(* Logix 5000 project; controller PRU vendor 1 type 14 code 107 rev 20.13; software revision 20.01; part 12 of 17 *)
(* tags used below, declared in another part *)
   AFI : BOOL;
   CR0_CON1_HTR1_GON : BOOL;   // ZONE 1 (L1,L2,L3)
   CR0_CON1_HTR1_LON : BOOL;   // AUTO LOGIC - ZONE 1 HEATER CONTACTOR
   CR1_CON2_HTR2_GON : BOOL;   // ZONE 2 (L1,L2,L3)
   CR1_CON2_HTR2_LON : BOOL;   // AUTO LOGIC - ZONE 2 HEATER CONTACTOR
   CR2_CON3_HTR3_GON : BOOL;   // ZONE 3 (L1,L2,L3)
   CR2_CON3_HTR3_LON : BOOL;   // AUTO LOGIC - ZONE 3 HEATER CONTACTOR
   CR3_CON4_HTR4_GON : BOOL;   // ZONE 4 (L1) ZONE 5 (L2) ZONE 6 (L3)
   CR3_CON4_HTR4_LON : BOOL;   // AUTO LOGIC - ZONES 4-6 HEATER CONTACTOR
   CR4_CON5_HTR5_GON : BOOL;   // ZONE 7 (L1) ZONE 8 (L2) ZONE 9 (L3)
   CR4_CON5_HTR5_LON : BOOL;   // AUTO LOGIC - ZONES 7-9 HEATER CONTACTOR
   CR5_CON1_SAFETY_GON : BOOL;
   CR5_CON1_SAFETY_LON : BOOL;
   CR6_CON2_SAFETY_GON : BOOL;
   CR6_CON2_SAFETY_LON : BOOL;
   CR8_VFD_DRYERR_GON : BOOL;
   CR8_VFD_DRYERR_LON : BOOL;
   ESR_CONTACT_1_ION : BOOL;
   ESR_CONTACT_2_ION : BOOL;
   ESR_RESET_PB_ION : BOOL;
   HMI_CR0_FORCE_OFF : BOOL;
   HMI_CR0_FORCE_ON : BOOL;
   HMI_CR10_FORCE_OFF : BOOL;
   HMI_CR10_FORCE_ON : BOOL;
   HMI_CR11_FORCE_OFF : BOOL;
   HMI_CR11_FORCE_ON : BOOL;
   HMI_CR12_FORCE_OFF : BOOL;
   HMI_CR12_FORCE_ON : BOOL;
   HMI_CR13_FORCE_OFF : BOOL;
   HMI_CR13_FORCE_ON : BOOL;
   HMI_CR14_FORCE_OFF : BOOL;   // Knife Gate 0621 force closed.
   HMI_CR14_FORCE_ON : BOOL;   // Knife Gate 0621 force open.
   HMI_CR15_FORCE_OFF : BOOL;   // Knife Gate 0621 force closed.
   HMI_CR15_FORCE_ON : BOOL;   // Knife Gate 0621 force open.
   HMI_CR16_FORCE_OFF : BOOL;
   HMI_CR16_FORCE_ON : BOOL;
   HMI_CR17_FORCE_OFF : BOOL;
   HMI_CR17_FORCE_ON : BOOL;
   HMI_CR19_FORCE_OFF : BOOL;
   HMI_CR19_FORCE_ON : BOOL;
   HMI_CR1_FORCE_OFF : BOOL;
   HMI_CR1_FORCE_ON : BOOL;
   HMI_CR2_FORCE_OFF : BOOL;
   HMI_CR2_FORCE_ON : BOOL;
   HMI_CR3_FORCE_OFF : BOOL;
   HMI_CR3_FORCE_ON : BOOL;
   HMI_CR4_FORCE_OFF : BOOL;
   HMI_CR4_FORCE_ON : BOOL;
   HMI_CR5_FORCE_OFF : BOOL;
   HMI_CR5_FORCE_ON : BOOL;
   HMI_CR6_FORCE_OFF : BOOL;
   HMI_CR6_FORCE_ON : BOOL;
   HMI_CR8_FORCE_OFF : BOOL;
   HMI_CR8_FORCE_ON : BOOL;
   HMI_CR9_FORCE_OFF : BOOL;
   HMI_CR9_FORCE_ON : BOOL;
   HMI_TE0101_FORCE_VALUE : INT;
   HMI_TE0101_FORCED : BOOL;
   HMI_TE0102_FORCE_VALUE : INT;
   HMI_TE0102_FORCED : BOOL;
   HMI_TE0103_FORCE_VALUE : INT;
   HMI_TE0103_FORCED : BOOL;
   HMI_TE0104_FORCE_VALUE : INT;
   HMI_TE0104_FORCED : BOOL;
   HMI_TE0105_FORCE_VALUE : INT;
   HMI_TE0105_FORCED : BOOL;
   HMI_TE0106_FORCE_VALUE : INT;
   HMI_TE0106_FORCED : BOOL;
   HMI_TE0107_FORCE_VALUE : INT;
   HMI_TE0107_FORCED : BOOL;
   HMI_TE0108_FORCE_VALUE : INT;
   HMI_TE0108_FORCED : BOOL;
   HMI_TE0109_FORCE_VALUE : DINT;
   HMI_TE0109_FORCED : BOOL;
   HMI_TE0110_FORCE_VALUE : DINT;
   HMI_TE0110_FORCED : BOOL;
   HMI_TE0111_FORCE_VALUE : DINT;
   HMI_TE0111_FORCED : BOOL;
   HMI_TE0112_FORCE_VALUE : DINT;
   HMI_TE0112_FORCED : BOOL;
   HMI_TE0113_FORCE_VALUE : DINT;
   HMI_TE0113_FORCED : BOOL;
   HMI_TE0114_FORCE_VALUE : DINT;
   HMI_TE0114_FORCED : BOOL;
   HMI_TE0115_FORCE_VALUE : DINT;
   HMI_TE0115_FORCED : BOOL;
   HMI_TE0116_FORCE_VALUE : DINT;
   HMI_TE0116_FORCED : BOOL;
   HMI_TE0117_FORCE_VALUE : DINT;
   HMI_TE0117_FORCED : BOOL;
   HMI_TE0118_FORCE_VALUE : DINT;
   HMI_TE0118_FORCED : BOOL;
   HMI_TE0119_FORCE_VALUE : DINT;
   HMI_TE0119_FORCED : BOOL;
   HMI_TE0120_FORCE_VALUE : DINT;
   HMI_TE0120_FORCED : BOOL;
   HMI_TE0121_FORCE_VALUE : DINT;
   HMI_TE0121_FORCED : BOOL;
   HMI_TE0122_FORCE_VALUE : DINT;
   HMI_TE0122_FORCED : BOOL;
   HMI_TE0123_FORCE_VALUE : DINT;
   HMI_TE0123_FORCED : BOOL;
   HMI_TE0124_FORCE_VALUE : DINT;
   HMI_TE0124_FORCED : BOOL;
   HMI_TE0125_FORCE_VALUE : DINT;
   HMI_TE0125_FORCED : BOOL;
   HMI_TE0126_FORCE_VALUE : DINT;
   HMI_TE0126_FORCED : BOOL;
   HMI_TE0127_FORCE_VALUE : DINT;
   HMI_TE0127_FORCED : BOOL;
   HMI_TE0128_FORCE_VALUE : DINT;
   HMI_TE0128_FORCED : BOOL;
   HMI_TE0129_FORCE_VALUE : DINT;
   HMI_TE0129_FORCED : BOOL;
   HMI_TE0130_FORCE_VALUE : DINT;
   HMI_TE0130_FORCED : BOOL;
   HMI_TE0201_FORCE_VALUE : DINT;
   HMI_TE0201_FORCED : BOOL;
   HMI_TE0202_FORCE_VALUE : DINT;
   HMI_TE0202_FORCED : BOOL;
   K6021_GO_CLOSE_GON : BOOL;
   K6021_GO_CLOSE_LON : BOOL;   // Knife Gate 6021 - Close Auto Logic
   K6021_GO_OPEN_GON : BOOL;
   K6021_GO_OPEN_LON : BOOL;   // Knife Gate 6021 - Open Auto Logic
   K6021_GO_STOP_GON : BOOL;
   K6022_GO_CLOSE_GON : BOOL;
   K6022_GO_CLOSE_LON : BOOL;
   K6022_GO_OPEN_GON : BOOL;
   K6022_GO_OPEN_LON : BOOL;
   K6022_GO_STOP_GON : BOOL;
   K6022_GO_STOP_LON : BOOL;
   KG021_SEQUENCER : INT;   // 1 = OPEN SV0201 2 = CLOSE SV0201 3 = OPEN KG021 4 = CLOSE KG021
   KG022_SEQUENCER : INT;   // 1 = OPEN SV0202 2 = CLOSE SV0202 3 = OPEN KG022 4 = CLOSE KG022
   PROCESS_SEQUENCER : INT;
   SHUTDOWN_PURGE_TIMER : TIMER;
   STARTUP_PURGE_TIMER : TIMER;
   SV0101 : BOOL;
   SV0101_LON : BOOL;
   SV0102 : BOOL;
   SV0102_LON : BOOL;
   SV0201 : BOOL;
   SV0201_LON : BOOL;
   SV0202 : BOOL;
   SV0202_LON : BOOL;
   SV0203 : BOOL;
   SV0203_LON : BOOL;
   TE0101 : REAL;
   TE0101_RAW : DINT;
   TE0102 : REAL;
   TE0102_RAW : DINT;
   TE0103 : REAL;
   TE0103_RAW : DINT;
   TE0104 : REAL;
   TE0104_RAW : DINT;
   TE0105 : REAL;
   TE0105_RAW : DINT;
   TE0106 : REAL;
   TE0106_RAW : DINT;
   TE0107 : REAL;
   TE0107_RAW : DINT;
   TE0108 : REAL;
   TE0108_RAW : DINT;
   TE0109 : REAL;
   TE0109_RAW : DINT;
   TE0110 : REAL;
   TE0110_RAW : DINT;
   TE0111 : REAL;
   TE0111_RAW : DINT;
   TE0112 : REAL;
   TE0112_RAW : DINT;
   TE0113 : REAL;
   TE0113_RAW : DINT;
   TE0114 : REAL;
   TE0114_RAW : DINT;
   TE0115 : REAL;
   TE0115_RAW : DINT;
   TE0116 : REAL;
   TE0116_RAW : DINT;
   TE0117 : REAL;
   TE0117_RAW : DINT;
   TE0118 : REAL;
   TE0118_RAW : DINT;
   TE0119 : REAL;
   TE0119_RAW : DINT;
   TE0120 : REAL;
   TE0120_RAW : DINT;
   TE0121 : REAL;
   TE0121_RAW : DINT;
   TE0122 : REAL;
   TE0122_RAW : DINT;
   TE0123 : REAL;
   TE0123_RAW : DINT;
   TE0124 : REAL;
   TE0124_RAW : DINT;
   TE0125 : REAL;
   TE0125_RAW : DINT;
   TE0126 : REAL;
   TE0126_RAW : DINT;
   TE0127 : REAL;
   TE0127_RAW : DINT;
   TE0128 : REAL;
   TE0128_RAW : DINT;
   TE0129 : REAL;
   TE0129_RAW : DINT;
   TE0130 : REAL;
   TE0130_RAW : DINT;
   TE0201 : REAL;
   TE0201_RAW : DINT;
   TE0202 : REAL;
   TE0202_RAW : DINT;
(* MainProgram, continued *)

ROUTINE G02_MAP_DIG_OUTPUTS   (* ladder *)
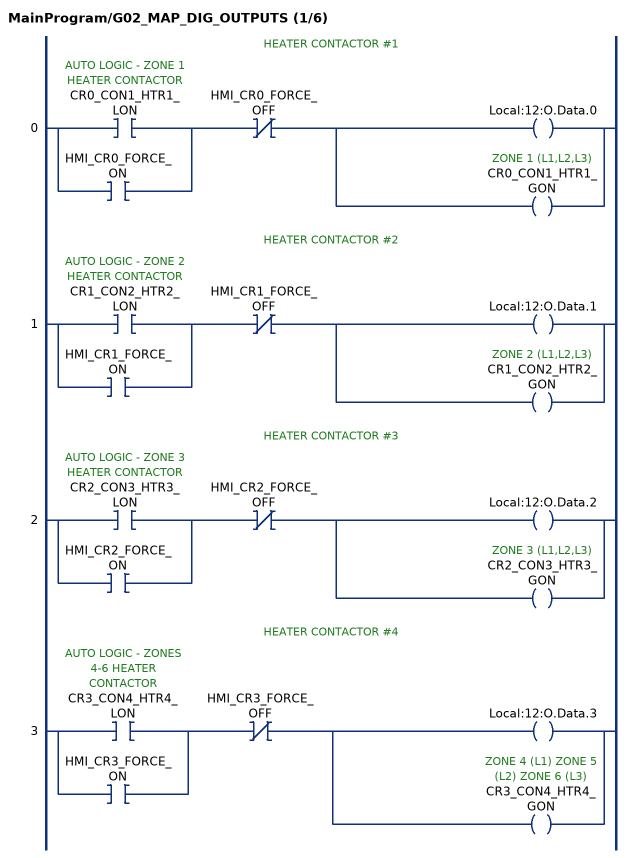
   // HEATER CONTACTOR #1
   0: [XIC(CR0_CON1_HTR1_LON) ,XIC(HMI_CR0_FORCE_ON) ]XIO(HMI_CR0_FORCE_OFF)[OTE(Local:12:O.Data.0) ,OTE(CR0_CON1_HTR1_GON) ];
   // HEATER CONTACTOR #2
   1: [XIC(CR1_CON2_HTR2_LON) ,XIC(HMI_CR1_FORCE_ON) ]XIO(HMI_CR1_FORCE_OFF)[OTE(Local:12:O.Data.1) ,OTE(CR1_CON2_HTR2_GON) ];
   // HEATER CONTACTOR #3
   2: [XIC(CR2_CON3_HTR3_LON) ,XIC(HMI_CR2_FORCE_ON) ]XIO(HMI_CR2_FORCE_OFF)[OTE(Local:12:O.Data.2) ,OTE(CR2_CON3_HTR3_GON) ];
   // HEATER CONTACTOR #4
   3: [XIC(CR3_CON4_HTR4_LON) ,XIC(HMI_CR3_FORCE_ON) ]XIO(HMI_CR3_FORCE_OFF)[OTE(Local:12:O.Data.3) ,OTE(CR3_CON4_HTR4_GON) ];
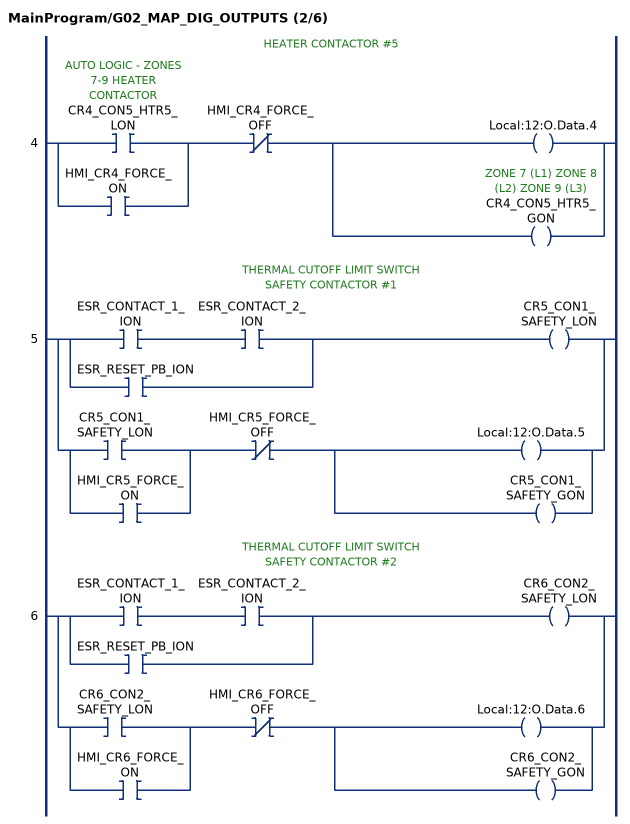
   // HEATER CONTACTOR #5
   4: [XIC(CR4_CON5_HTR5_LON) ,XIC(HMI_CR4_FORCE_ON) ]XIO(HMI_CR4_FORCE_OFF)[OTE(Local:12:O.Data.4) ,OTE(CR4_CON5_HTR5_GON) ];
   // THERMAL CUTOFF LIMIT SWITCH
   // SAFETY CONTACTOR #1
   5: [[XIC(ESR_CONTACT_1_ION) XIC(ESR_CONTACT_2_ION) ,XIC(ESR_RESET_PB_ION) ] OTE(CR5_CON1_SAFETY_LON) ,[XIC(CR5_CON1_SAFETY_LON) ,XIC(HMI_CR5_FORCE_ON) ] XIO(HMI_CR5_FORCE_OFF) [OTE(Local:12:O.Data.5) ,OTE(CR5_CON1_SAFETY_GON) ] ];
   // THERMAL CUTOFF LIMIT SWITCH
   // SAFETY CONTACTOR #2
   6: [[XIC(ESR_CONTACT_1_ION) XIC(ESR_CONTACT_2_ION) ,XIC(ESR_RESET_PB_ION) ] OTE(CR6_CON2_SAFETY_LON) ,[XIC(CR6_CON2_SAFETY_LON) ,XIC(HMI_CR6_FORCE_ON) ] XIO(HMI_CR6_FORCE_OFF) [OTE(Local:12:O.Data.6) ,OTE(CR6_CON2_SAFETY_GON) ] ];
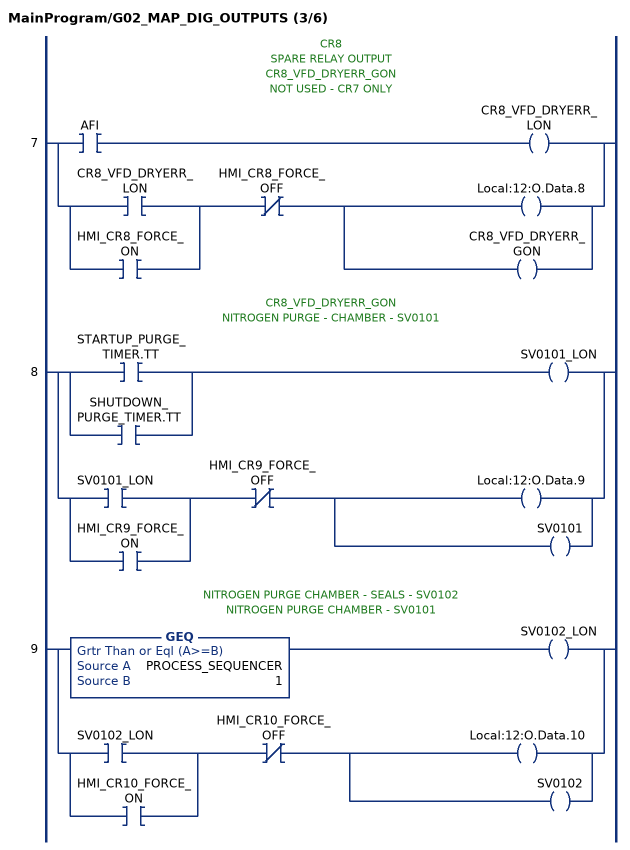
   // CR8
   // SPARE RELAY OUTPUT
   // CR8_VFD_DRYERR_GON
   // NOT USED - CR7 ONLY
   7: [XIC(AFI) OTE(CR8_VFD_DRYERR_LON) ,[XIC(CR8_VFD_DRYERR_LON) ,XIC(HMI_CR8_FORCE_ON) ] XIO(HMI_CR8_FORCE_OFF) [OTE(Local:12:O.Data.8) ,OTE(CR8_VFD_DRYERR_GON) ] ];
   // CR8_VFD_DRYERR_GON
   // NITROGEN PURGE - CHAMBER - SV0101
   8: [[XIC(STARTUP_PURGE_TIMER.TT) ,XIC(SHUTDOWN_PURGE_TIMER.TT) ] OTE(SV0101_LON) ,[XIC(SV0101_LON) ,XIC(HMI_CR9_FORCE_ON) ] XIO(HMI_CR9_FORCE_OFF) [OTE(Local:12:O.Data.9) ,OTE(SV0101) ] ];
   // NITROGEN PURGE CHAMBER - SEALS - SV0102
   // NITROGEN PURGE CHAMBER - SV0101
   9: [GEQ(PROCESS_SEQUENCER,1) OTE(SV0102_LON) ,[XIC(SV0102_LON) ,XIC(HMI_CR10_FORCE_ON) ] XIO(HMI_CR10_FORCE_OFF) [OTE(Local:12:O.Data.10) ,OTE(SV0102) ] ];
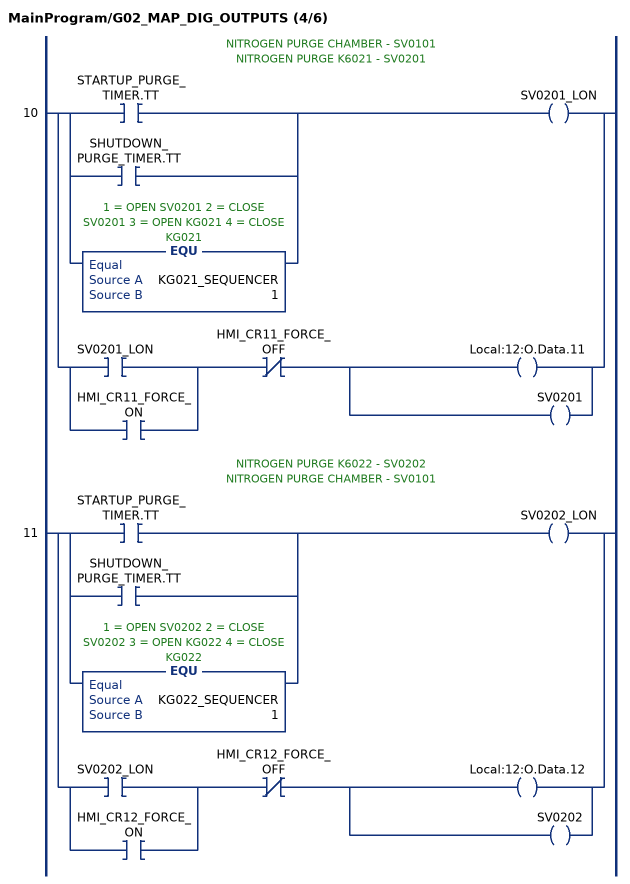
   // NITROGEN PURGE CHAMBER - SV0101
   // NITROGEN PURGE K6021 - SV0201
   10: [[XIC(STARTUP_PURGE_TIMER.TT) ,XIC(SHUTDOWN_PURGE_TIMER.TT) ,EQU(KG021_SEQUENCER,1) ] OTE(SV0201_LON) ,[XIC(SV0201_LON) ,XIC(HMI_CR11_FORCE_ON) ] XIO(HMI_CR11_FORCE_OFF) [OTE(Local:12:O.Data.11) ,OTE(SV0201) ] ];
   // NITROGEN PURGE K6022 - SV0202
   // NITROGEN PURGE CHAMBER - SV0101
   11: [[XIC(STARTUP_PURGE_TIMER.TT) ,XIC(SHUTDOWN_PURGE_TIMER.TT) ,EQU(KG022_SEQUENCER,1) ] OTE(SV0202_LON) ,[XIC(SV0202_LON) ,XIC(HMI_CR12_FORCE_ON) ] XIO(HMI_CR12_FORCE_OFF) [OTE(Local:12:O.Data.12) ,OTE(SV0202) ] ];
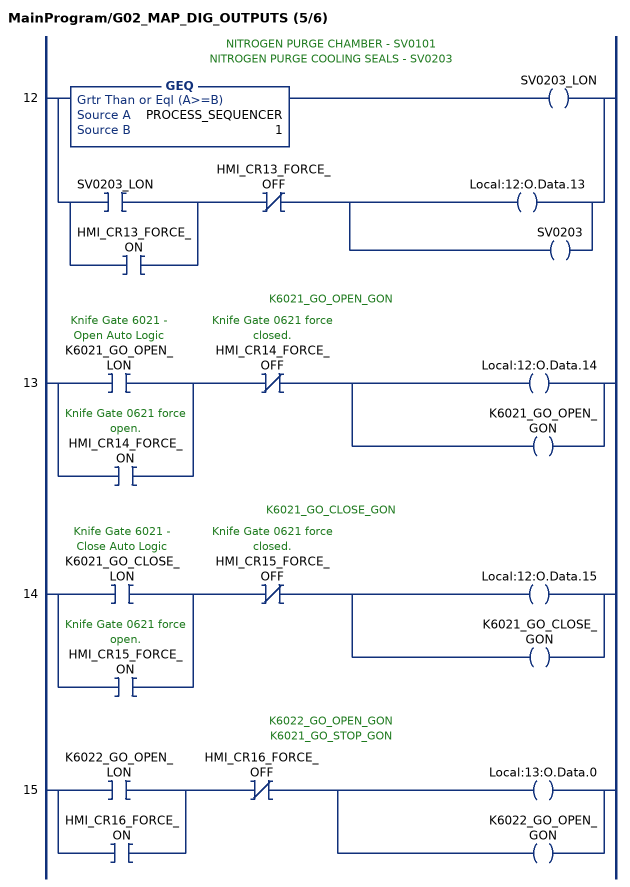
   // NITROGEN PURGE CHAMBER - SV0101
   // NITROGEN PURGE COOLING SEALS - SV0203
   12: [GEQ(PROCESS_SEQUENCER,1) OTE(SV0203_LON) ,[XIC(SV0203_LON) ,XIC(HMI_CR13_FORCE_ON) ] XIO(HMI_CR13_FORCE_OFF) [OTE(Local:12:O.Data.13) ,OTE(SV0203) ] ];
   // K6021_GO_OPEN_GON
   13: [XIC(K6021_GO_OPEN_LON) ,XIC(HMI_CR14_FORCE_ON) ]XIO(HMI_CR14_FORCE_OFF)[OTE(Local:12:O.Data.14) ,OTE(K6021_GO_OPEN_GON) ];
   // K6021_GO_CLOSE_GON
   14: [XIC(K6021_GO_CLOSE_LON) ,XIC(HMI_CR15_FORCE_ON) ]XIO(HMI_CR15_FORCE_OFF)[OTE(Local:12:O.Data.15) ,OTE(K6021_GO_CLOSE_GON) ];
   // K6022_GO_OPEN_GON
   // K6021_GO_STOP_GON
   15: [XIC(K6022_GO_OPEN_LON) ,XIC(HMI_CR16_FORCE_ON) ]XIO(HMI_CR16_FORCE_OFF)[OTE(Local:13:O.Data.0) ,OTE(K6022_GO_OPEN_GON) ];
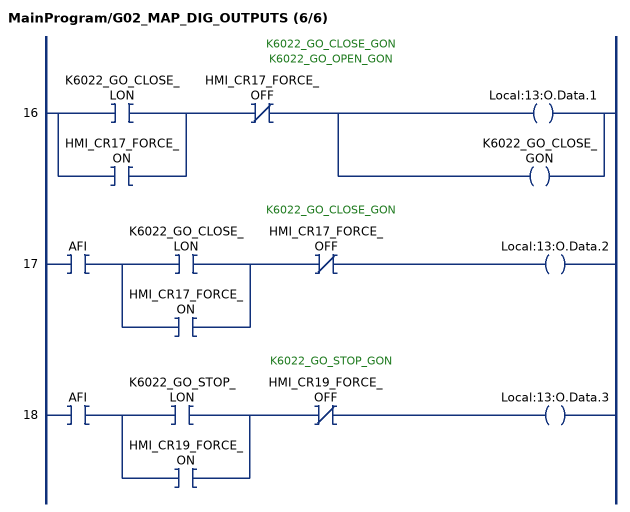
   // K6022_GO_CLOSE_GON
   // K6022_GO_OPEN_GON
   16: [XIC(K6022_GO_CLOSE_LON) ,XIC(HMI_CR17_FORCE_ON) ]XIO(HMI_CR17_FORCE_OFF)[OTE(Local:13:O.Data.1) ,OTE(K6022_GO_CLOSE_GON) ];
   // K6022_GO_CLOSE_GON
   17: XIC(AFI)[XIC(K6022_GO_CLOSE_LON) ,XIC(HMI_CR17_FORCE_ON) ]XIO(HMI_CR17_FORCE_OFF)OTE(Local:13:O.Data.2);
   // K6022_GO_STOP_GON
   18: XIC(AFI)[XIC(K6022_GO_STOP_LON) ,XIC(HMI_CR19_FORCE_ON) ]XIO(HMI_CR19_FORCE_OFF)OTE(Local:13:O.Data.3);
END_ROUTINE

ROUTINE G03_MAP_THERMOCOUPLES   (* ladder *)
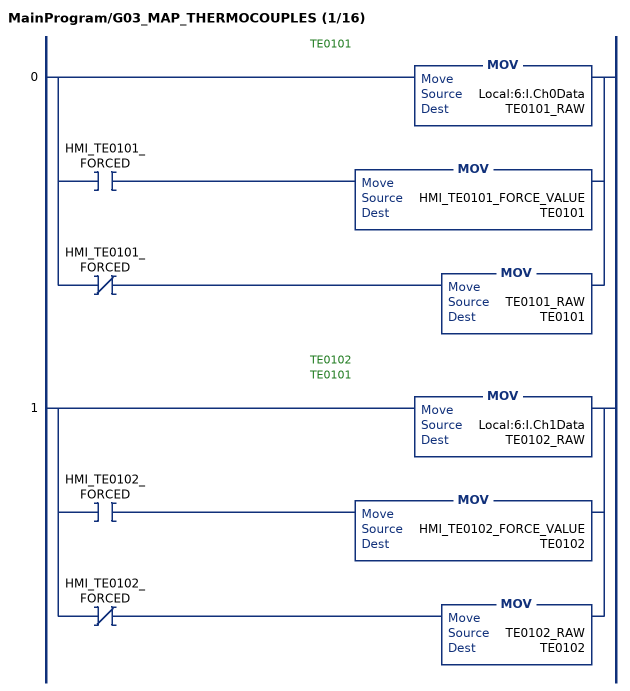
   // TE0101
   0: [MOV(Local:6:I.Ch0Data,TE0101_RAW) ,XIC(HMI_TE0101_FORCED) MOV(HMI_TE0101_FORCE_VALUE,TE0101) ,XIO(HMI_TE0101_FORCED) MOV(TE0101_RAW,TE0101) ];
   // TE0102
   // TE0101
   1: [MOV(Local:6:I.Ch1Data,TE0102_RAW) ,XIC(HMI_TE0102_FORCED) MOV(HMI_TE0102_FORCE_VALUE,TE0102) ,XIO(HMI_TE0102_FORCED) MOV(TE0102_RAW,TE0102) ];
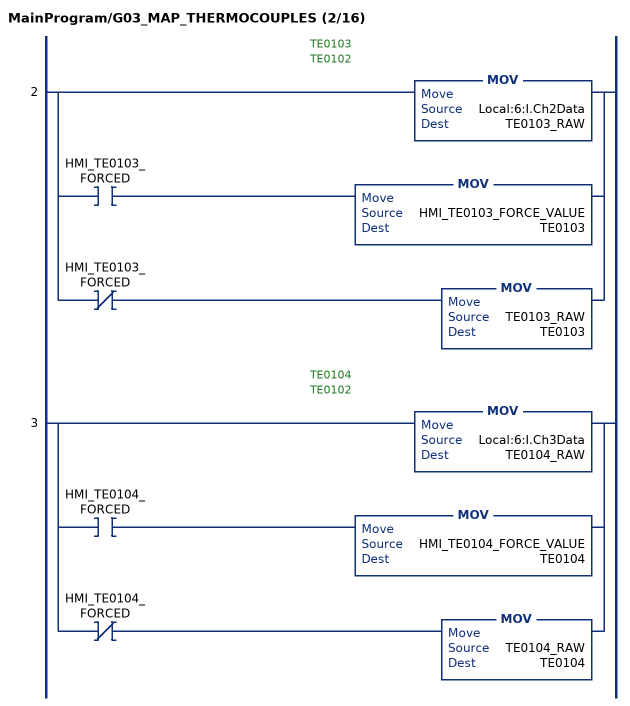
   // TE0103
   // TE0102
   2: [MOV(Local:6:I.Ch2Data,TE0103_RAW) ,XIC(HMI_TE0103_FORCED) MOV(HMI_TE0103_FORCE_VALUE,TE0103) ,XIO(HMI_TE0103_FORCED) MOV(TE0103_RAW,TE0103) ];
   // TE0104
   // TE0102
   3: [MOV(Local:6:I.Ch3Data,TE0104_RAW) ,XIC(HMI_TE0104_FORCED) MOV(HMI_TE0104_FORCE_VALUE,TE0104) ,XIO(HMI_TE0104_FORCED) MOV(TE0104_RAW,TE0104) ];
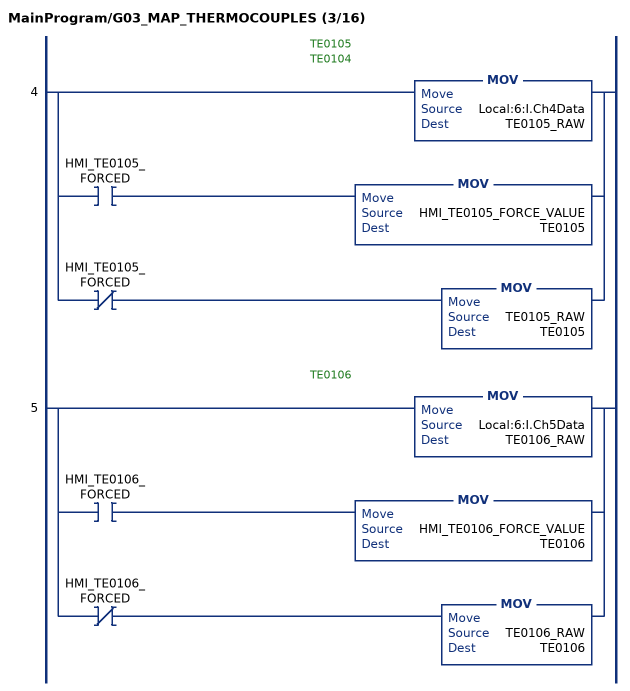
   // TE0105
   // TE0104
   4: [MOV(Local:6:I.Ch4Data,TE0105_RAW) ,XIC(HMI_TE0105_FORCED) MOV(HMI_TE0105_FORCE_VALUE,TE0105) ,XIO(HMI_TE0105_FORCED) MOV(TE0105_RAW,TE0105) ];
   // TE0106
   5: [MOV(Local:6:I.Ch5Data,TE0106_RAW) ,XIC(HMI_TE0106_FORCED) MOV(HMI_TE0106_FORCE_VALUE,TE0106) ,XIO(HMI_TE0106_FORCED) MOV(TE0106_RAW,TE0106) ];
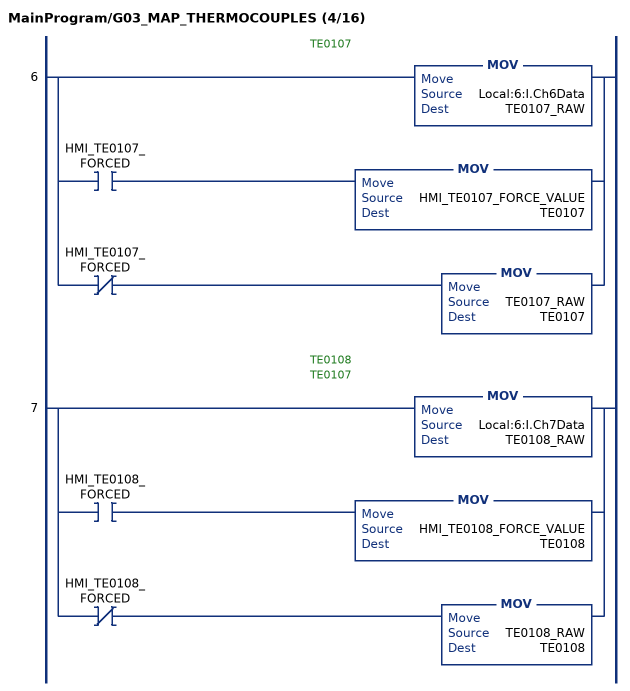
   // TE0107
   6: [MOV(Local:6:I.Ch6Data,TE0107_RAW) ,XIC(HMI_TE0107_FORCED) MOV(HMI_TE0107_FORCE_VALUE,TE0107) ,XIO(HMI_TE0107_FORCED) MOV(TE0107_RAW,TE0107) ];
   // TE0108
   // TE0107
   7: [MOV(Local:6:I.Ch7Data,TE0108_RAW) ,XIC(HMI_TE0108_FORCED) MOV(HMI_TE0108_FORCE_VALUE,TE0108) ,XIO(HMI_TE0108_FORCED) MOV(TE0108_RAW,TE0108) ];
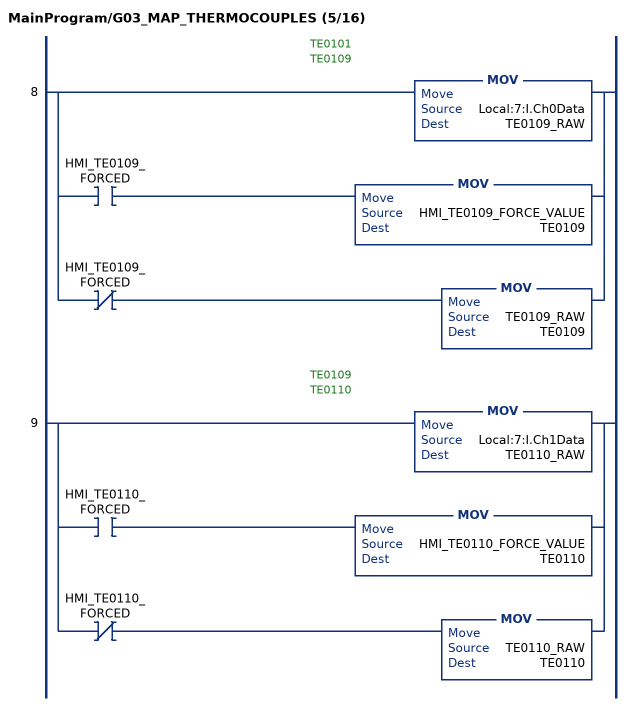
   // TE0101
   // TE0109
   8: [MOV(Local:7:I.Ch0Data,TE0109_RAW) ,XIC(HMI_TE0109_FORCED) MOV(HMI_TE0109_FORCE_VALUE,TE0109) ,XIO(HMI_TE0109_FORCED) MOV(TE0109_RAW,TE0109) ];
   // TE0109
   // TE0110
   9: [MOV(Local:7:I.Ch1Data,TE0110_RAW) ,XIC(HMI_TE0110_FORCED) MOV(HMI_TE0110_FORCE_VALUE,TE0110) ,XIO(HMI_TE0110_FORCED) MOV(TE0110_RAW,TE0110) ];
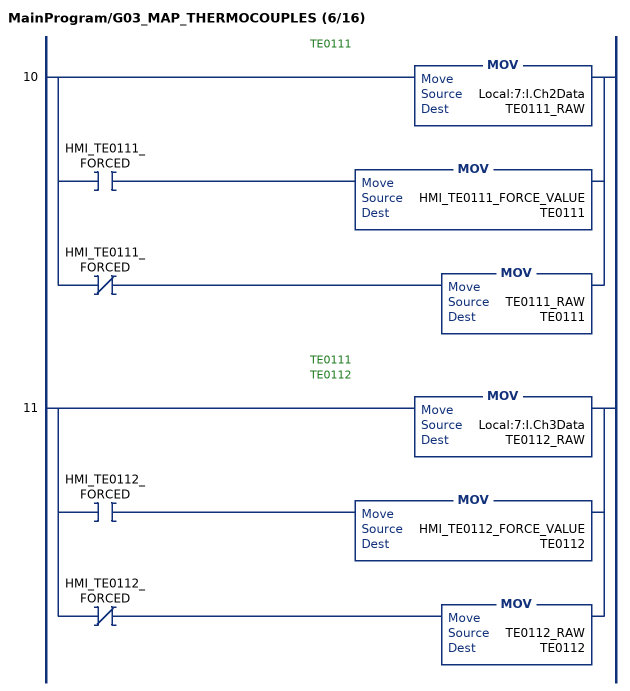
   // TE0111
   10: [MOV(Local:7:I.Ch2Data,TE0111_RAW) ,XIC(HMI_TE0111_FORCED) MOV(HMI_TE0111_FORCE_VALUE,TE0111) ,XIO(HMI_TE0111_FORCED) MOV(TE0111_RAW,TE0111) ];
   // TE0111
   // TE0112
   11: [MOV(Local:7:I.Ch3Data,TE0112_RAW) ,XIC(HMI_TE0112_FORCED) MOV(HMI_TE0112_FORCE_VALUE,TE0112) ,XIO(HMI_TE0112_FORCED) MOV(TE0112_RAW,TE0112) ];
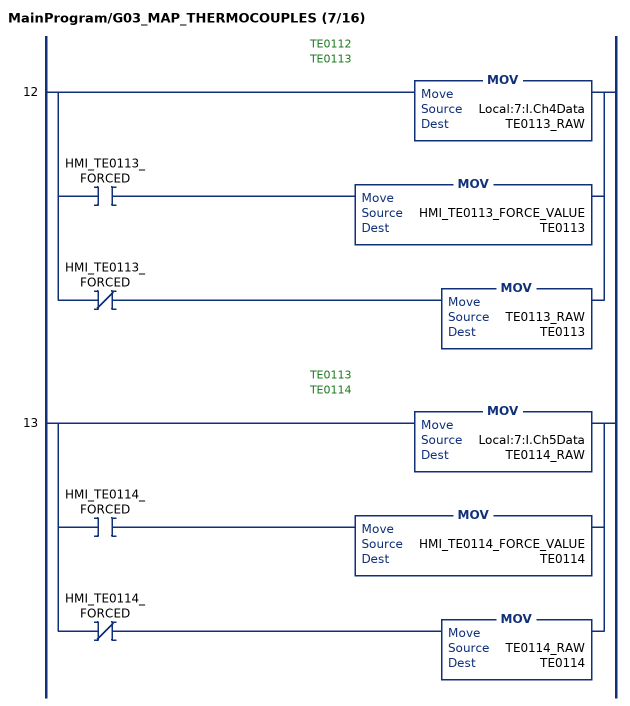
   // TE0112
   // TE0113
   12: [MOV(Local:7:I.Ch4Data,TE0113_RAW) ,XIC(HMI_TE0113_FORCED) MOV(HMI_TE0113_FORCE_VALUE,TE0113) ,XIO(HMI_TE0113_FORCED) MOV(TE0113_RAW,TE0113) ];
   // TE0113
   // TE0114
   13: [MOV(Local:7:I.Ch5Data,TE0114_RAW) ,XIC(HMI_TE0114_FORCED) MOV(HMI_TE0114_FORCE_VALUE,TE0114) ,XIO(HMI_TE0114_FORCED) MOV(TE0114_RAW,TE0114) ];
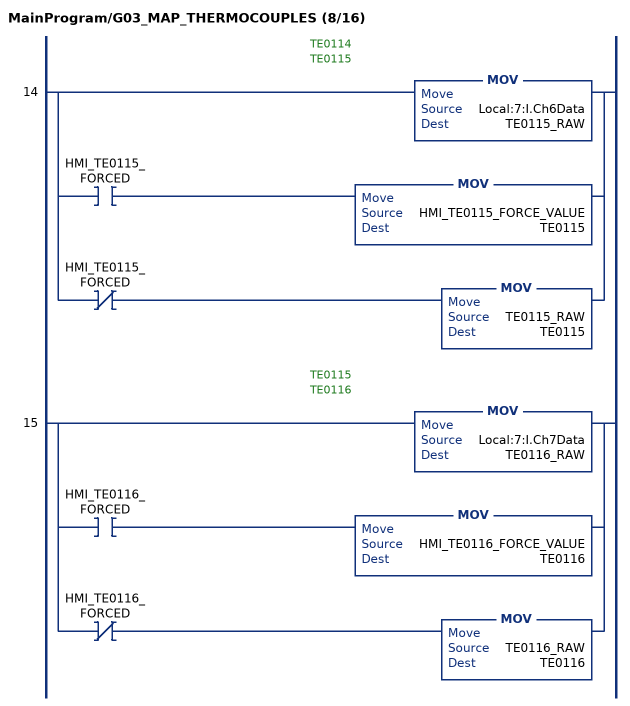
   // TE0114
   // TE0115
   14: [MOV(Local:7:I.Ch6Data,TE0115_RAW) ,XIC(HMI_TE0115_FORCED) MOV(HMI_TE0115_FORCE_VALUE,TE0115) ,XIO(HMI_TE0115_FORCED) MOV(TE0115_RAW,TE0115) ];
   // TE0115
   // TE0116
   15: [MOV(Local:7:I.Ch7Data,TE0116_RAW) ,XIC(HMI_TE0116_FORCED) MOV(HMI_TE0116_FORCE_VALUE,TE0116) ,XIO(HMI_TE0116_FORCED) MOV(TE0116_RAW,TE0116) ];
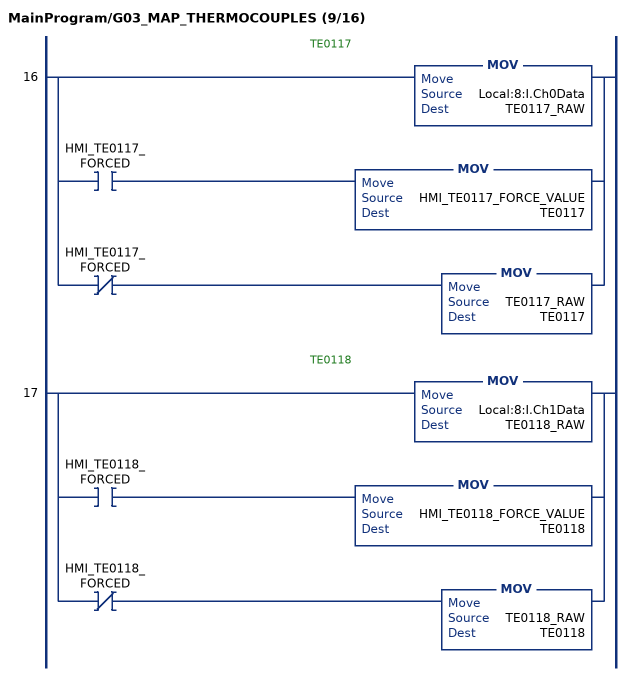
   // TE0117
   16: [MOV(Local:8:I.Ch0Data,TE0117_RAW) ,XIC(HMI_TE0117_FORCED) MOV(HMI_TE0117_FORCE_VALUE,TE0117) ,XIO(HMI_TE0117_FORCED) MOV(TE0117_RAW,TE0117) ];
   // TE0118
   17: [MOV(Local:8:I.Ch1Data,TE0118_RAW) ,XIC(HMI_TE0118_FORCED) MOV(HMI_TE0118_FORCE_VALUE,TE0118) ,XIO(HMI_TE0118_FORCED) MOV(TE0118_RAW,TE0118) ];
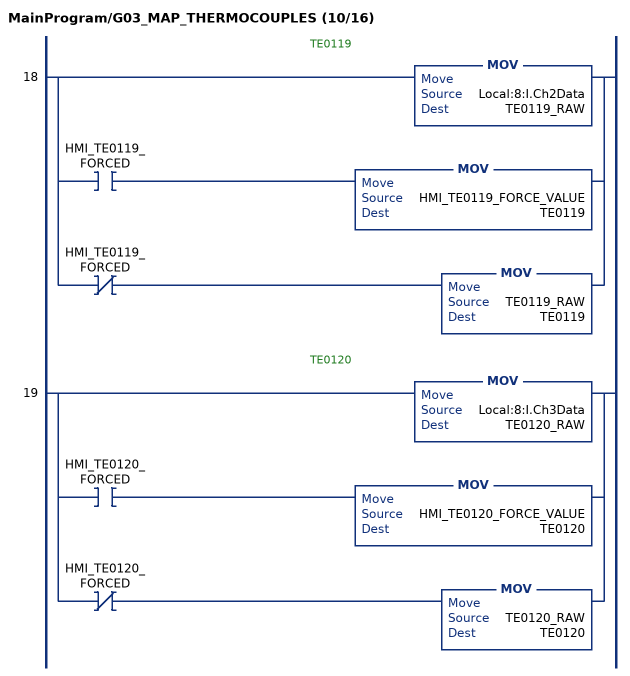
   // TE0119
   18: [MOV(Local:8:I.Ch2Data,TE0119_RAW) ,XIC(HMI_TE0119_FORCED) MOV(HMI_TE0119_FORCE_VALUE,TE0119) ,XIO(HMI_TE0119_FORCED) MOV(TE0119_RAW,TE0119) ];
   // TE0120
   19: [MOV(Local:8:I.Ch3Data,TE0120_RAW) ,XIC(HMI_TE0120_FORCED) MOV(HMI_TE0120_FORCE_VALUE,TE0120) ,XIO(HMI_TE0120_FORCED) MOV(TE0120_RAW,TE0120) ];
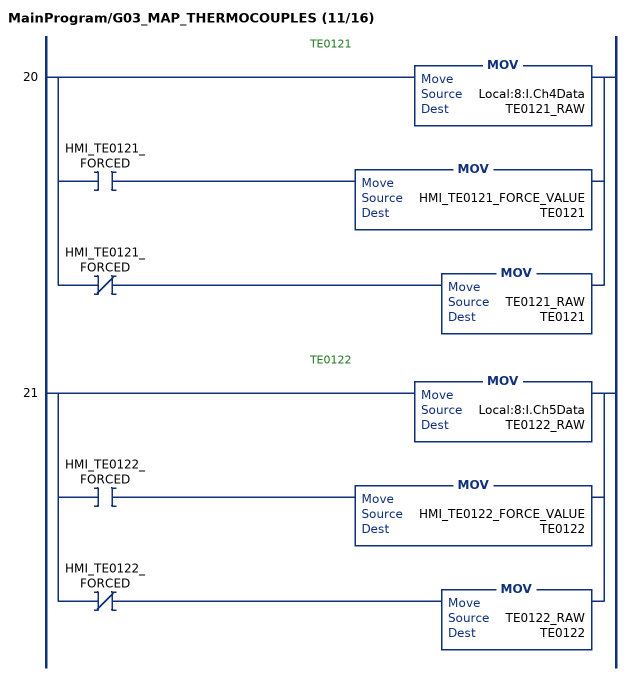
   // TE0121
   20: [MOV(Local:8:I.Ch4Data,TE0121_RAW) ,XIC(HMI_TE0121_FORCED) MOV(HMI_TE0121_FORCE_VALUE,TE0121) ,XIO(HMI_TE0121_FORCED) MOV(TE0121_RAW,TE0121) ];
   // TE0122
   21: [MOV(Local:8:I.Ch5Data,TE0122_RAW) ,XIC(HMI_TE0122_FORCED) MOV(HMI_TE0122_FORCE_VALUE,TE0122) ,XIO(HMI_TE0122_FORCED) MOV(TE0122_RAW,TE0122) ];
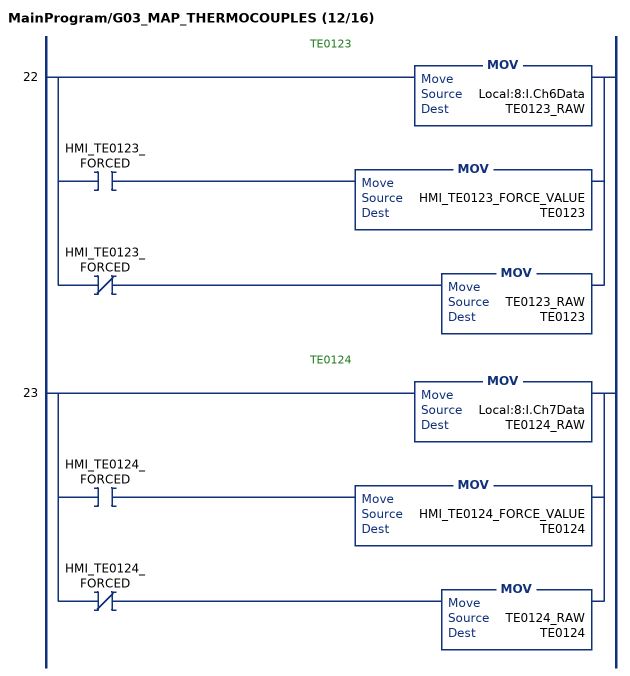
   // TE0123
   22: [MOV(Local:8:I.Ch6Data,TE0123_RAW) ,XIC(HMI_TE0123_FORCED) MOV(HMI_TE0123_FORCE_VALUE,TE0123) ,XIO(HMI_TE0123_FORCED) MOV(TE0123_RAW,TE0123) ];
   // TE0124
   23: [MOV(Local:8:I.Ch7Data,TE0124_RAW) ,XIC(HMI_TE0124_FORCED) MOV(HMI_TE0124_FORCE_VALUE,TE0124) ,XIO(HMI_TE0124_FORCED) MOV(TE0124_RAW,TE0124) ];
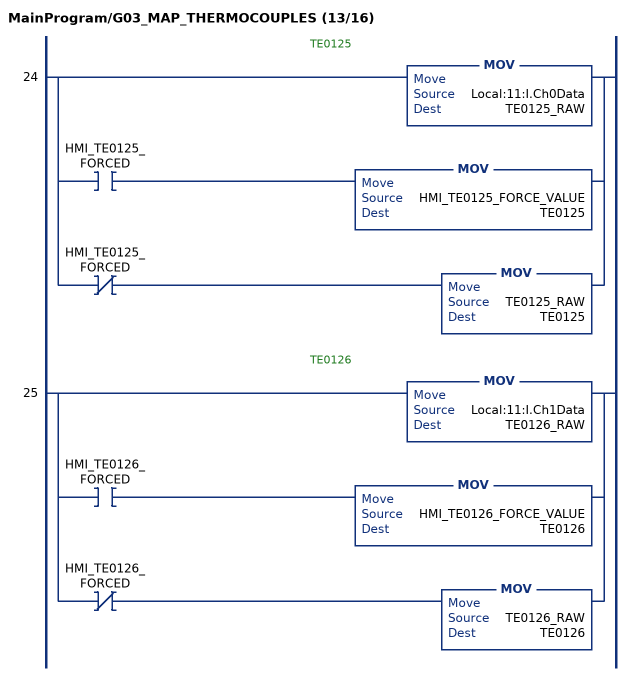
   // TE0125
   24: [MOV(Local:11:I.Ch0Data,TE0125_RAW) ,XIC(HMI_TE0125_FORCED) MOV(HMI_TE0125_FORCE_VALUE,TE0125) ,XIO(HMI_TE0125_FORCED) MOV(TE0125_RAW,TE0125) ];
   // TE0126
   25: [MOV(Local:11:I.Ch1Data,TE0126_RAW) ,XIC(HMI_TE0126_FORCED) MOV(HMI_TE0126_FORCE_VALUE,TE0126) ,XIO(HMI_TE0126_FORCED) MOV(TE0126_RAW,TE0126) ];
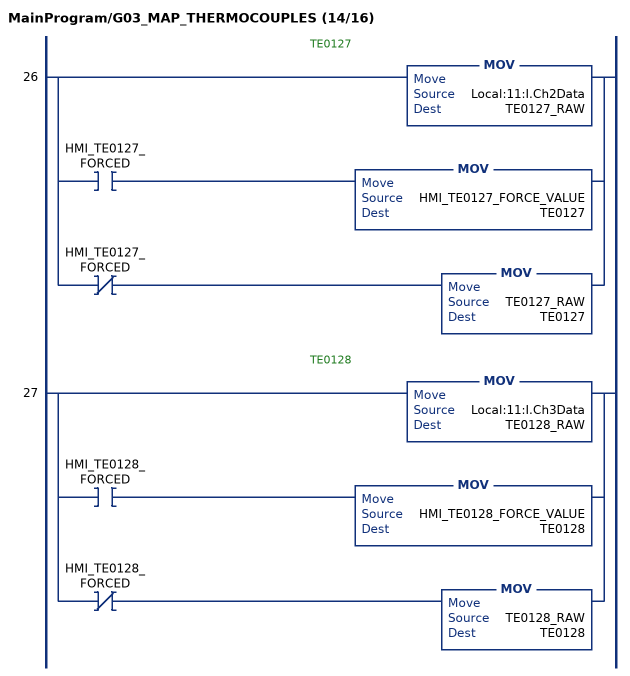
   // TE0127
   26: [MOV(Local:11:I.Ch2Data,TE0127_RAW) ,XIC(HMI_TE0127_FORCED) MOV(HMI_TE0127_FORCE_VALUE,TE0127) ,XIO(HMI_TE0127_FORCED) MOV(TE0127_RAW,TE0127) ];
   // TE0128
   27: [MOV(Local:11:I.Ch3Data,TE0128_RAW) ,XIC(HMI_TE0128_FORCED) MOV(HMI_TE0128_FORCE_VALUE,TE0128) ,XIO(HMI_TE0128_FORCED) MOV(TE0128_RAW,TE0128) ];
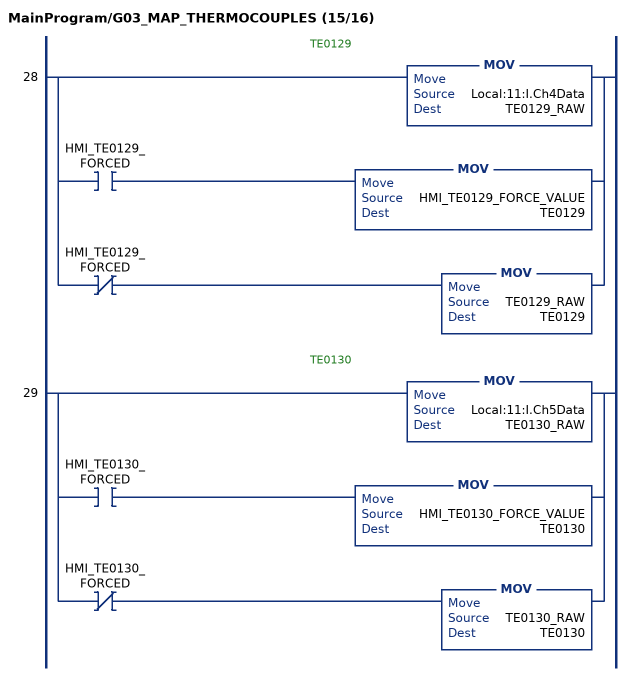
   // TE0129
   28: [MOV(Local:11:I.Ch4Data,TE0129_RAW) ,XIC(HMI_TE0129_FORCED) MOV(HMI_TE0129_FORCE_VALUE,TE0129) ,XIO(HMI_TE0129_FORCED) MOV(TE0129_RAW,TE0129) ];
   // TE0130
   29: [MOV(Local:11:I.Ch5Data,TE0130_RAW) ,XIC(HMI_TE0130_FORCED) MOV(HMI_TE0130_FORCE_VALUE,TE0130) ,XIO(HMI_TE0130_FORCED) MOV(TE0130_RAW,TE0130) ];
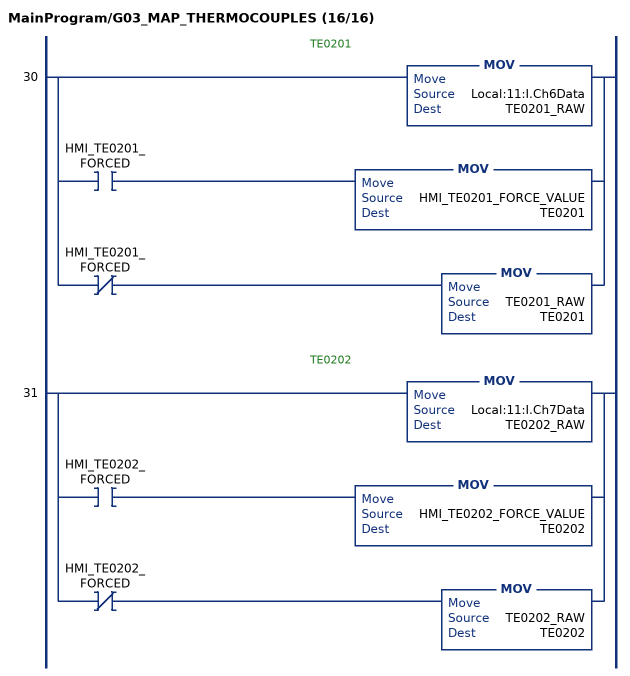
   // TE0201
   30: [MOV(Local:11:I.Ch6Data,TE0201_RAW) ,XIC(HMI_TE0201_FORCED) MOV(HMI_TE0201_FORCE_VALUE,TE0201) ,XIO(HMI_TE0201_FORCED) MOV(TE0201_RAW,TE0201) ];
   // TE0202
   31: [MOV(Local:11:I.Ch7Data,TE0202_RAW) ,XIC(HMI_TE0202_FORCED) MOV(HMI_TE0202_FORCE_VALUE,TE0202) ,XIO(HMI_TE0202_FORCED) MOV(TE0202_RAW,TE0202) ];
END_ROUTINE
